FUNCTION_BLOCK FB_StXPlanarData IMPLEMENTS ITF_StXPlanarData
VAR_INPUT
	fbMover								: REFERENCE TO MC_PlanarMover;
END_VAR
VAR_OUTPUT
	ST_XPLANAR_DATA						: ST_XPLANAR_DATA;
END_VAR
VAR
	ActPosition							: MoverVector;
	ActVelocity							: MoverVector;
	SetPosition							: MoverVector;
	SetVelocity							: MoverVector;
END_VAR

ActPosition := fbMover.MCTOPLC.ACT.ActPos;
ActVelocity := fbMover.MCTOPLC.ACT.ActVelo;
SetPosition := fbMover.MCTOPLC.SET.SetPos;
SetVelocity := fbMover.MCTOPLC.SET.SetVelo;

//General
ST_XPLANAR_DATA.uiState := THIS^.GetState;
ST_XPLANAR_DATA.bState_Error := THIS^.GetStateError;
ST_XPLANAR_DATA.uiMoverErrorID := THIS^.GetErrorID;
ST_XPLANAR_DATA.uliTimeStamp := THIS^.GetTimeStamp;
ST_XPLANAR_DATA.uiDemoState := THIS^.GetDemoState;

// ActPosition
ST_XPLANAR_DATA.lrActPosition_x := THIS^.GetActPosition_x;
ST_XPLANAR_DATA.lrActPosition_y := THIS^.GetActPosition_y;
ST_XPLANAR_DATA.lrActPosition_z := THIS^.GetActPosition_z;
ST_XPLANAR_DATA.lrActPosition_a := THIS^.GetActPosition_a;
ST_XPLANAR_DATA.lrActPosition_b := THIS^.GetActPosition_b;
ST_XPLANAR_DATA.lrActPosition_c := THIS^.GetActPosition_c;
// SetPosition
ST_XPLANAR_DATA.lrSetPosition_x := THIS^.GetSetPosition_x;
ST_XPLANAR_DATA.lrSetPosition_y := THIS^.GetSetPosition_y;
ST_XPLANAR_DATA.lrSetPosition_z := THIS^.GetSetPosition_z;
ST_XPLANAR_DATA.lrSetPosition_a := THIS^.GetSetPosition_a;
ST_XPLANAR_DATA.lrSetPosition_b := THIS^.GetSetPosition_b;
ST_XPLANAR_DATA.lrSetPosition_c := THIS^.GetSetPosition_c;
// ActVelocity
ST_XPLANAR_DATA.lrActVelocity_x := THIS^.GetActVelocity_x;
ST_XPLANAR_DATA.lrActVelocity_y := THIS^.GetActVelocity_y;
ST_XPLANAR_DATA.lrActVelocity_z := THIS^.GetActVelocity_z;
ST_XPLANAR_DATA.lrActVelocity_a := THIS^.GetActVelocity_a;
ST_XPLANAR_DATA.lrActVelocity_b := THIS^.GetActVelocity_b;
ST_XPLANAR_DATA.lrActVelocity_c := THIS^.GetActVelocity_c;
// SetVelocity
ST_XPLANAR_DATA.lrSetVelocity_x := THIS^.GetSetVelocity_x;
ST_XPLANAR_DATA.lrSetVelocity_y := THIS^.GetSetVelocity_y;
ST_XPLANAR_DATA.lrSetVelocity_z := THIS^.GetSetVelocity_z;
ST_XPLANAR_DATA.lrSetVelocity_a := THIS^.GetSetVelocity_a;
ST_XPLANAR_DATA.lrSetVelocity_b := THIS^.GetSetVelocity_b;
ST_XPLANAR_DATA.lrSetVelocity_c := THIS^.GetSetVelocity_c;

{warning 'add method implementation '}
METHOD GetActPosition_a : LREAL
GetActPosition_a := ActPosition.a;
END_METHOD

{warning 'add method implementation '}
METHOD GetActPosition_b : LREAL
GetActPosition_b := ActPosition.b;
END_METHOD

{warning 'add method implementation '}
METHOD GetActPosition_c : LREAL
GetActPosition_c := ActPosition.c;
END_METHOD

{warning 'add method implementation '}
METHOD GetActPosition_x : LREAL
GetActPosition_x := ActPosition.x;
END_METHOD

{warning 'add method implementation '}
METHOD GetActPosition_y : LREAL
GetActPosition_y := ActPosition.y;
END_METHOD

{warning 'add method implementation '}
METHOD GetActPosition_z : LREAL
GetActPosition_z := ActPosition.z;
END_METHOD

{warning 'add method implementation '}
METHOD GetActVelocity_a : LREAL
GetActVelocity_a := ActVelocity.a;
END_METHOD

{warning 'add method implementation '}
METHOD GetActVelocity_b : LREAL
GetActVelocity_b := ActVelocity.b;
END_METHOD

{warning 'add method implementation '}
METHOD GetActVelocity_c : LREAL
GetActVelocity_c := ActVelocity.c;
END_METHOD

{warning 'add method implementation '}
METHOD GetActVelocity_x : LREAL
GetActVelocity_x := ActVelocity.x;
END_METHOD

{warning 'add method implementation '}
METHOD GetActVelocity_y : LREAL
GetActVelocity_y := ActVelocity.y;
END_METHOD

{warning 'add method implementation '}
METHOD GetActVelocity_z : LREAL
GetActVelocity_z := ActVelocity.z;
END_METHOD

{warning 'add method implementation '}
METHOD GetDemoState : UINT
END_METHOD

{warning 'add method implementation '}
METHOD GetErrorID : UINT
END_METHOD

{warning 'add method implementation '}
METHOD GetSetPosition_a : LREAL
END_METHOD

{warning 'add method implementation '}
METHOD GetSetPosition_b : LREAL
END_METHOD

{warning 'add method implementation '}
METHOD GetSetPosition_c : LREAL
END_METHOD

{warning 'add method implementation '}
METHOD GetSetPosition_x : LREAL
END_METHOD

{warning 'add method implementation '}
METHOD GetSetPosition_y : LREAL
END_METHOD

{warning 'add method implementation '}
METHOD GetSetPosition_z : LREAL
END_METHOD

{warning 'add method implementation '}
METHOD GetSetVelocity_a : LREAL
END_METHOD

{warning 'add method implementation '}
METHOD GetSetVelocity_b : LREAL
END_METHOD

{warning 'add method implementation '}
METHOD GetSetVelocity_c : LREAL
END_METHOD

{warning 'add method implementation '}
METHOD GetSetVelocity_x : LREAL
END_METHOD

{warning 'add method implementation '}
METHOD GetSetVelocity_y : LREAL
END_METHOD

{warning 'add method implementation '}
METHOD GetSetVelocity_z : LREAL
END_METHOD

{warning 'add method implementation '}
METHOD GetState : UINT
END_METHOD

{warning 'add method implementation '}
METHOD GetStateError : BOOL
END_METHOD

{warning 'add method implementation '}
METHOD GetTimeStamp : ULINT
END_METHOD

END_FUNCTION_BLOCK

(* stored: Version 1.1.0.1, ProductVersion 3.1.4024.11
   POU FB_StXPlanarData: Id {e003ed92-715c-4594-ac45-4de666637235}, SpecialFunc None
   Folder ActPosition: Id {eea02ac7-7096-4ce3-a72a-6877ed6e563c}
   Folder ActVelocity: Id {f4a11e78-bd1f-40ad-9067-2a28fb52fe5a}
   Folder General: Id {476f7462-91e6-448a-ab5c-2c0a7b46a39b}
   Folder SetPosition: Id {164555b5-f2a4-4feb-b096-d2312bb7395b}
   Folder SetVelocity: Id {9d0436d7-118c-4db9-9606-27dae6bd2400}
   Method GetActPosition_a: Id {9a778402-58b4-4955-bb88-2ffe698e137a}
   Method GetActPosition_b: Id {c774a813-43e6-4053-88f8-582dc006ec0b}
   Method GetActPosition_c: Id {74a03d50-96bb-43da-bb8f-aecb208cd273}
   Method GetActPosition_x: Id {24b82646-1eff-413d-8ef0-06e8b110c47a}
   Method GetActPosition_y: Id {498a8a25-79ac-4310-9cdf-74ac93d4a9d9}
   Method GetActPosition_z: Id {29e79948-2467-4fc6-a18a-4546e26d2b88}
   Method GetActVelocity_a: Id {d8e46300-3496-4713-bcdb-61361e230700}
   Method GetActVelocity_b: Id {b613af1c-1956-4214-9e85-ec1bf500203d}
   Method GetActVelocity_c: Id {0cd1627f-3764-417f-90b7-df87be4408cc}
   Method GetActVelocity_x: Id {9650db03-e53b-4f10-859b-6c7ee8c40b90}
   Method GetActVelocity_y: Id {2dedd5c1-e486-413a-bd49-08a583fed0ac}
   Method GetActVelocity_z: Id {e9096169-6f32-40bb-bc43-fb8410b419ed}
   Method GetDemoState: Id {251c8cfe-1315-4be2-a2fb-71a394881ab0}
   Method GetErrorID: Id {c35b675d-ed6d-4f10-982e-9c6e08f51dce}
   Method GetSetPosition_a: Id {4ee85e73-9f2e-4768-a440-d5853c7f8e91}
   Method GetSetPosition_b: Id {cf4c213a-ce80-4202-8353-6286d758f551}
   Method GetSetPosition_c: Id {8bfc7cfc-6c36-4665-a18a-63aa90bfabed}
   Method GetSetPosition_x: Id {17cca9dd-db20-47ca-a178-90add1dc4083}
   Method GetSetPosition_y: Id {ed3e25b5-afd3-4df7-a69d-e900b96edd6f}
   Method GetSetPosition_z: Id {d970f4a7-0367-4cbb-b307-ae36e44350ce}
   Method GetSetVelocity_a: Id {f7a85b30-5a8c-46c8-83ea-47b360fe48ea}
   Method GetSetVelocity_b: Id {1b578392-5607-4be2-953f-9b6c48c797ee}
   Method GetSetVelocity_c: Id {8734e2cc-eeeb-4401-817d-a50a52b03733}
   Method GetSetVelocity_x: Id {489f13f5-ff62-499a-a612-db4e01a7b4f8}
   Method GetSetVelocity_y: Id {ab2c021b-86ea-4217-b89f-9673337b45b5}
   Method GetSetVelocity_z: Id {8db3b38f-69bc-4ebe-a003-9f27e34c1cdf}
   Method GetState: Id {4fd6b760-ba87-42e8-9784-da983bc25b59}
   Method GetStateError: Id {d9a1e248-b7d3-4769-a43b-18fbc07f617c}
   Method GetTimeStamp: Id {d1244442-9456-477a-8000-398db107258c} *)
